SUBAPPLICATION Ventilsteuerung_Uebung_031 (* LED Strip *)
  (* Standard: 61499-2 *)
  (* Version 1.0, 2023-10-23, franz *)
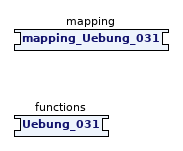
  SUBAPPS
    mapping : mapping_Uebung_031;
    functions : Uebung_031;
  END_SUBAPPS
END_SUBAPPLICATION
